{attribute 'linkalways'} 
{attribute 'no_explicit_call' := 'This FB is a CLASS and must be accessed using methods or properties'}
{attribute 'enable_dynamic_creation'}
FUNCTION_BLOCK FINAL LE_UDINT EXTENDS Node
VAR
	in1 : _UDINT(0);
	in2 : _UDINT(0);
	out : _BOOL(FALSE);
END_VAR

METHOD PUBLIC Clone : I_Node
VAR
	pNode : POINTER TO LE_UDINT;
END_VAR
pNode := __NEW(LE_UDINT);
Clone := pNode^;
END_METHOD

METHOD FB_init : BOOL
VAR_INPUT
	bInitRetains : BOOL; // if TRUE, the retain variables are initialized (warm start / cold start)
	bInCopyCode : BOOL;  // if TRUE, the instance afterwards gets moved into the copy code (online change)
END_VAR
AddInput('in1',THIS^.in1);
AddInput('in2',THIS^.in2);
AddOutput('out', THIS^.out);
END_METHOD

METHOD PROTECTED OnExecute
VAR
END_VAR
out.Value := in1.Value <= in2.Value;
END_METHOD

END_FUNCTION_BLOCK

(* stored: Version 1.1.0.1, ProductVersion 3.1.4024.15
   POU LE_UDINT: Id {54202dfb-f4af-4889-8466-bc168e27ba9e}, SpecialFunc None
   Folder Constructor: Id {be30b83e-0eac-4ae6-a2f1-781e810ba1ae}
   Method Clone: Id {4fb2d97a-10a5-47ba-abe8-0d86764b278c}
   Method FB_init: Id {c0f98d30-6f88-47b5-becb-8d097d583e28}
   Method OnExecute: Id {0246772d-f9ad-4673-8ef3-5c96140d9fa2} *)
